TYPE ST_ModuleControl :
STRUCT
	bEnableDisable		: BOOL; // CMD 1A
	rSetOutputVoltage	: REAL;	// CMD 1C
	rSetOutputCurrent	: REAL;	// CMD 1C
	
	
	
	
END_STRUCT
END_TYPE

(* stored: Version 1.1.0.1, ProductVersion 3.1.4026.18
   DUT ST_ModuleControl: Id {64c7cf45-4eff-4a61-b3fa-ebd1459e7879} *)
